FUNCTION_BLOCK FB_Controller_PID EXTENDS FB_Controller_PI
VAR_INPUT
END_VAR
VAR_OUTPUT
END_VAR
VAR
	_Tv	: TIME;
	_Td	: TIME;
END_VAR

// Executes the controller and returns the control output.
METHOD Execute
VAR_OUTPUT
	controllerOutput	: LREAL;	// Controller result
END_VAR
PID.fTd := THIS^.TimeToSeconds(_Td);
PID.fTv := THIS^.TimeToSeconds(_Tv);
SUPER^.Execute();
END_METHOD

// Gets or sets the damping time
PROPERTY Td : TIME
GET
Td := _Td;
END_GET
SET
_Td := Td;
END_SET
END_PROPERTY

// Gets or sets the derivative action time.
PROPERTY Tv : TIME
GET
Tv := _Tv;
END_GET
SET
_Tv := Tv;
END_SET
END_PROPERTY

END_FUNCTION_BLOCK

(* stored: Version 1.1.0.1, ProductVersion 3.1.4024.14
   POU FB_Controller_PID: Id {ddcebbcd-d47c-0f0e-0c61-24b7ea616d14}, SpecialFunc None
   Method Execute: Id {5755f55c-df20-0ac1-0586-238435c7f8b3}
   Property Td: Id {4d538e31-f527-07e9-3126-88c859123ebf}
   Get Get: Id {60a48e5d-e736-0e9d-01d3-715ee8923fc9}
   Set Set: Id {b9687066-0c3e-0a78-24d7-c07166245b02}
   Property Tv: Id {665a33c5-c470-0c36-1d85-15b8e645be29}
   Get Get: Id {26a93eef-aee0-0ea6-369c-1b191f252200}
   Set Set: Id {3b64c8ed-0cb3-0451-0953-02a3242224ad} *)
